(* CoDeSys 2.3.9.62 project: SemaforoGRAFCET MP.pro *)
(* Libraries: Standard.lib 2.6.14 10:37:46, IecSfc.lib 2.6.14 10:37:46 *)

(* Global variable list: Global_Variables *)
VAR_GLOBAL

 (* Entradas *)
	M: BOOL;
        P:BOOL;

      (*Salidas*)
	Rojo: BOOL;    	(* Luz roja*)
	Amarillo:BOOL;	(* Luz amarilla *)
	Verde:BOOL;		(* Luz verde *)

END_VAR

(* POU PLC_PRG, SFC *)
PROGRAM PLC_PRG
VAR
    (* declaración  de contadores *)
	CONTA: CTU;
END_VAR
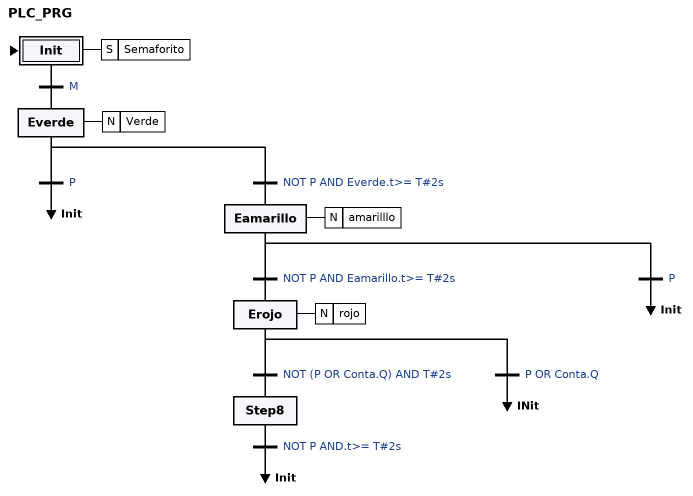
INITIAL_STEP Init:
	Semaforito(S);
END_STEP
TRANSITION FROM Init TO Everde := M;
END_TRANSITION
STEP Everde:
	Verde(N);
END_STEP
TRANSITION FROM Everde TO Init := P;
END_TRANSITION
TRANSITION FROM Everde TO Eamarillo := NOT P AND Everde.t>= T#2s;
END_TRANSITION
STEP Eamarillo:
	amarilllo(N);
END_STEP
TRANSITION FROM Eamarillo TO Erojo := NOT P AND Eamarillo.t>= T#2s;
END_TRANSITION
TRANSITION FROM Eamarillo TO Init := P;
END_TRANSITION
STEP Erojo:
	rojo(N);
END_STEP
TRANSITION FROM Erojo TO Step8 := NOT (P OR Conta.Q) AND T#2s;
END_TRANSITION
TRANSITION FROM Erojo TO INit := P OR Conta.Q;
END_TRANSITION
STEP Step8:
END_STEP
TRANSITION FROM Step8 TO Init := NOT P AND.t>= T#2s;
END_TRANSITION
END_PROGRAM
ACTION Semaforito:

END_ACTION

(* Visualisation SemaforoSimple
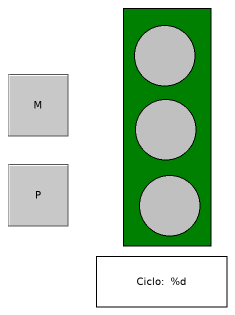
ellipse at (156,41)-(217,102): alarm colour if Rojo
ellipse at (157,115)-(218,176): alarm colour if Amarillo
ellipse at (161,191)-(222,252): alarm colour if Verde
rectangle at (118,272)-(249,323): text "Ciclo:  %d"; shows PLC_PRG.CONTA.CV
button at (30,90)-(90,152): text "M"; taps M
button at (30,180)-(90,242): text "P"; taps P
1 more shapes without text or variables
*)
